// TIA Portal V19 export
DATA_BLOCK "iPALARMS"   // DB500
AUTHOR : CH
FAMILY : Aktina
NAME : Faults
// stored: AutoNumber false, InstanceOfName pALARMS, InstanceOfType FB
"pALARMS"
   // VAR
   //    "75sf1" : "AFB_AlarmAckn";
   // END_VAR
BEGIN
   "75sf1".trigger := FALSE;
   "75sf1".release := TRUE;
   "75sf1".ctrlpoint := TRUE;
   "75sf1".enackn := TRUE;
   "75sf1".ensiren := TRUE;
   "75sf1".p100ms := TRUE;
   "75sf1".generalackn := FALSE;
   "75sf1".reset := FALSE;
   "75sf1".mute := FALSE;
   "75sf1".delay := 0.5;
   "75sf1".plcackn := FALSE;
   "75sf1".alarm := FALSE;
   "75sf1".siren := FALSE;
   "75sf1".hmiackn := FALSE;
   "75sf1".i.setup.en := TRUE;
   "75sf1".i.setup.spon := 0.0;
   "75sf1".i.don.countup := FALSE;
   "75sf1".i.don.sp := 5;
   "75sf1".i.don.actual := 0;
   "75sf1".i.don.end := FALSE;
   "75sf1".i.status.plcackn := FALSE;
   "75sf1".i.status.alarm := FALSE;
   "75sf1".i.status.siren := FALSE;
END_DATA_BLOCK
